Staubli VAL3: loadAction.pgx

program loadAction(string x_sPallet, num x_nOffset)
  local num l_nPos
  local num l_nSize[3]
  local string l_sAction
begin
  //
  // get the actual position
  //
  call getPalletPos(x_sPallet,l_nPos)
  // PLANE CONDITION
  // loook for the z quote
  l_sAction=pt:tTraj[sTrajCycle].sAction[l_nPos%pt:tTraj[sTrajCycle].nZ]
  if (l_nPos+1)%(pt:tTraj[sTrajCycle].nY*pt:tTraj[sTrajCycle].nX)==0 and l_sAction!=""
    // show the string
    cycleStatus:sToShow="CALL PALLET PROG "+l_sAction
    // SET THE JUMP for the CALL..
    cycleStatus:bCALL=true
    // NB use the session field
    cycleStatus:iToSuperV.sType="PROG"
    cycleStatus:iToSuperV.sData=l_sAction
    use:bUseRefresh=true
  endIf
end
